// TwinCAT 3 PLC project superimposed_plc_demo
// ProgramVersion: 3.1.4023.0
// CompilerDefines: VISU_USEWSTRING
// libraries:
//   Tc2_MC2, * (Beckhoff Automation GmbH)
//   Tc2_Standard, * (Beckhoff Automation GmbH)
//   Tc2_System, * (Beckhoff Automation GmbH)
//   Tc3_Module, * (Beckhoff Automation GmbH)
//   VisuSymbols,3.5.10.0,System
// project tree:
//   / GlobalTextList.TcGTLO, PlcTask.TcTTO, VISU_TASK.TcTTO, 视图管理器.TcVMO (not stored)
//   POUs/ MAIN.TcPOU
//   POUs/superimpose/ superimpose.TcPOU, SuperimposedActural.TcDUT
//   VISUs/ superimposed.TcVIS
// real-time tasks:
//   TASK PlcTask: cycle T#10ms, priority 20, ADS port 350
//   TASK VISU_TASK: cycle T#200000us, priority 30, ADS port 351
// motion (NC):
//   TASK NC-Task 1 SAF: cycle T#2ms, priority 4, ADS port 501
//   TASK NC-Task 1 SVB: cycle T#10ms, priority 8, ADS port 511
//   AXIS Axis 1 (id 1)
//     OtherSettings: AllowMotionCmdToSlave=true
//     encoder EncType=1
//     drive DrvType=5
//       Analog: TorqueSetpointScale=10, ScaleFactorActTorque=0.1
//       TimeComp: TaskDelayCycles=1
//     controller CtrType=1
//       CtrPara: PriorControlFactor=1
//         Observer: BandWidth=20
//   AXIS Axis 2 (id 2)
//     OtherSettings: AllowMotionCmdToSlave=true
//     encoder EncType=1
//     drive DrvType=5
//       Analog: TorqueSetpointScale=10, ScaleFactorActTorque=0.1
//       TimeComp: TaskDelayCycles=1
//     controller CtrType=1
//       CtrPara: PriorControlFactor=1
//         Observer: BandWidth=20
// variable links:
//   superimposed_plc_demo/superimposed_plc_demo Instance <-> NC-Task 1 SAF/Axes/Axis 1
//     PlcTask Inputs/superimpose.axis1.NcToPlc <-> Outputs/ToPlc
//     PlcTask Outputs/superimpose.axis1.PlcToNc <-> Inputs/FromPlc
//   superimposed_plc_demo/superimposed_plc_demo Instance <-> NC-Task 1 SAF/Axes/Axis 2
//     PlcTask Inputs/superimpose.axis2.NcToPlc <-> Outputs/ToPlc
//     PlcTask Outputs/superimpose.axis2.PlcToNc <-> Inputs/FromPlc

CONFIGURATION superimposed_plc_demo
    RESOURCE PLC ON TwinCAT3
        TASK PlcTask(INTERVAL := T#10ms, PRIORITY := 20);
        TASK VISU_TASK(INTERVAL := T#200000us, PRIORITY := 30);
        PROGRAM MAIN WITH PlcTask : MAIN;
        PROGRAM VisuElems_Visu_Prg WITH VISU_TASK : VisuElems.Visu_Prg;
    END_RESOURCE
END_CONFIGURATION

// ---- POUs/superimpose/SuperimposedActural.TcDUT
TYPE SuperimposedActural :
STRUCT
	Done               : BOOL;
    Busy               : BOOL;
    Active             : BOOL;
    CommandAborted     : BOOL;
    Error              : BOOL;
    ErrorID            : UDINT;
	Warning            : BOOL;
    WarningID          : UDINT;
    ActualVelocityDiff : LREAL;
    ActualDistance     : LREAL;
    ActualLength       : LREAL;
    ActualAcceleration : LREAL;
    ActualDeceleration : LREAL;
END_STRUCT
END_TYPE

// ---- POUs/MAIN.TcPOU
PROGRAM MAIN
VAR

END_VAR

superimpose();

END_PROGRAM

// ---- POUs/superimpose/superimpose.TcPOU
PROGRAM superimpose
VAR
	axis1 						: AXIS_REF;
	axis2 						: AXIS_REF;
			
	mcSetPosition1 				: MC_SetPosition;
	mcSetPosition2 				: MC_SetPosition;
	setPositionOutput1 			: ST_McOutputs;
	setPositionOutput2 			: ST_McOutputs;
	shouldSetPosition			: BOOL;
	
	mcMoveVelocity1				: MC_MoveVelocity;
	mcMoveVelocity2				: MC_MoveVelocity;
	moveVelocityOutput1			: ST_McOutputs;
	moveVelocityOutput2			: ST_McOutputs;
	shouldMoveVelocity			: BOOL;
	
	mcMoveSuperImposed			: MC_MoveSuperImposed;
	moveSuperImposedOutput		: SuperimposedActural;
	
	positionDiff: LREAL;
END_VAR

(*
axis1();
axis2();
*)

power();
checkSetPosition();
checkMoveVelocity();
checkToSuperimpose();

mcMoveSuperImposed.Execute:= shouldMoveVelocity;
mcMoveSuperImposed.Mode := 2;
mcMoveSuperImposed.Distance := 300;
mcMoveSuperImposed.VelocityDiff := 500;
mcMoveSuperImposed.VelocityProcess := 700;
mcMoveSuperImposed.Length := 1000;

positionDiff:= axis2.NcToPlc.SetPos - axis1.NcToPlc.SetPos;
mcSetPosition1.Execute := shouldSetPosition;
mcSetPosition2.Execute := shouldSetPosition;
mcMoveVelocity1.Execute := shouldMoveVelocity;
mcMoveVelocity2.Execute := shouldMoveVelocity;

ACTION checkMoveVelocity:
mcMoveVelocity1(
	Axis:= axis1, 
	Execute:= shouldMoveVelocity, 
	Velocity:= 200, 
	Acceleration:= , 
	Deceleration:= , 
	Jerk:= , 
	Direction:= 1, 
	BufferMode:= , 
	Options:= , 
	InVelocity=> moveVelocityOutput1.Done, 
	Busy=> moveVelocityOutput1.Busy, 
	Active=> moveVelocityOutput1.Active, 
	CommandAborted=> moveVelocityOutput1.CommandAborted, 
	Error=> moveVelocityOutput1.Error, 
	ErrorID=> moveVelocityOutput1.ErrorID);
	
mcMoveVelocity2(
	Axis:= axis2, 
	Execute:= shouldMoveVelocity, 
	Velocity:= 200, 
	Acceleration:= , 
	Deceleration:= , 
	Jerk:= , 
	Direction:= 1, 
	BufferMode:= , 
	Options:= , 
	InVelocity=> moveVelocityOutput2.Done, 
	Busy=> moveVelocityOutput2.Busy, 
	Active=> moveVelocityOutput2.Active, 
	CommandAborted=> moveVelocityOutput2.CommandAborted, 
	Error=> moveVelocityOutput2.Error, 
	ErrorID=> moveVelocityOutput2.ErrorID);
END_ACTION

ACTION checkSetPosition:
mcSetPosition1(
	Axis:= axis1, 
	Execute:= mcSetPosition1.Execute, 
	Position:= 0, 
	Mode:= , 
	Options:= , 
	Done=> setPositionOutput1.Done, 
	Busy=> setPositionOutput1.Busy, 
	Error=> setPositionOutput1.Error, 
	ErrorID=> setPositionOutput1.ErrorID);
	
mcSetPosition2(
	Axis:= axis2, 
	Execute:= mcSetPosition2.Execute, 
	Position:= 1800, 
	Mode:= , 
	Options:= , 
	Done=> setPositionOutput2.Done, 
	Busy=> setPositionOutput2.Busy, 
	Error=> setPositionOutput2.Error, 
	ErrorID=> setPositionOutput2.ErrorID);
END_ACTION

ACTION checkToSuperimpose:
mcMoveSuperImposed(
	Axis:= axis1, 
	Execute:= mcMoveSuperImposed.Execute, 
	Mode:= mcMoveSuperImposed.Mode, 
	Distance:= mcMoveSuperImposed.Distance, 
	VelocityDiff:= mcMoveSuperImposed.VelocityDiff, 
	Acceleration:= mcMoveSuperImposed.Acceleration, 
	Deceleration:= mcMoveSuperImposed.Deceleration, 
	Jerk:= mcMoveSuperImposed.Jerk, 
	VelocityProcess:= mcMoveSuperImposed.VelocityProcess, 
	Length:= mcMoveSuperImposed.Length, 
	Options:= , 
	Done=> moveSuperImposedOutput.Done, 
	Busy=> moveSuperImposedOutput.Busy, 
	Active=> moveSuperImposedOutput.Active, 
	CommandAborted=> moveSuperImposedOutput.CommandAborted, 
	Error=> moveSuperImposedOutput.Error, 
	ErrorID=> moveSuperImposedOutput.ErrorID, 
	Warning=> moveSuperImposedOutput.Warning, 
	WarningId=> moveSuperImposedOutput.WarningID, 
	ActualVelocityDiff=> moveSuperImposedOutput.ActualVelocityDiff, 
	ActualDistance=> moveSuperImposedOutput.ActualDistance, 
	ActualLength=> moveSuperImposedOutput.ActualLength, 
	ActualAcceleration=> moveSuperImposedOutput.ActualAcceleration, 
	ActualDeceleration=> moveSuperImposedOutput.ActualDeceleration);
END_ACTION

ACTION power:
axis1.PlcToNc.ControlDWord:=7;
axis1.PlcToNc.Override:=1000000;
axis2.PlcToNc.ControlDWord:=7;
axis2.PlcToNc.Override:=1000000;
END_ACTION

END_PROGRAM

// ---- GlobalTextList.TcGTLO
TEXTLIST GlobalTextList
  963 = 'move super'
  38 = 'set position'
END_TEXTLIST

// ---- VISUs/superimposed.TcVIS
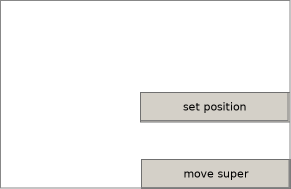
VISUALIZATION superimposed  // 291x189
    Button (140,92 150x30), "set position", colour toggle: superimpose.shouldSetPosition
        tap superimpose.shouldSetPosition
    Button (141,159 150x30), "move super", colour toggle: superimpose.shouldMoveVelocity
        tap superimpose.shouldMoveVelocity
END_VISUALIZATION
